TYPE ST_MV_JAVA_Zustand :
STRUCT
	Beheizung_Aktiv	: BOOL;
	Betrieb			: BOOL;
	Kommunikation	: BOOL;
	Warnung			: BOOL;
	Warnung_Code	: WORD;
	Stoerung		: BOOL;
	Stoerung_Code	: WORD;
	Beheizung_VL_XS_Temp	: REAL;
END_STRUCT
END_TYPE

(* stored: Version 1.1.0.1, ProductVersion 3.1.4024.9
   DUT ST_MV_JAVA_Zustand: Id {7c5eb825-5137-4984-be9d-5315594d9c59} *)
